FUNCTION_BLOCK FIFO_StatsAggregate
VAR_INPUT
	Overwrite: BOOL;
	pFIFO: POINTER TO StatsAggregateFIFOBuffer;
	in: StatsAggregateRecord;
END_VAR

VAR_OUTPUT
	Err: BOOL;
	Count: DINT;
	Full: BOOL;
	out: StatsAggregateRecord;
END_VAR

VAR
	Head	: UDINT;
	Tail	: UDINT;
	Idx		: UDINT;
END_VAR

ACTION INIT:
Idx := pFIFO^.Size * SIZEOF(in);
MEMSET(ADR(pFIFO^.Buffer[0]), 0, Idx);
MEMSET(ADR(in), 0, SIZEOF(in));
MEMSET(ADR(out), 0, SIZEOF(out));
Count := 0;
Head := 0;
Tail := 0;
Full := 0;
Err := 0;
END_ACTION

ACTION LOAD:
Err := 0;
IF (Full AND Overwrite) OR NOT Full THEN
	pFIFO^.Buffer[Head] := in;
	Head := Head + 1;
	IF Head = pFIFO^.Size THEN
		Head := 0;
	END_IF
	IF Full THEN
		Tail := Tail + 1;
		IF Tail = pFIFO^.Size THEN
			Tail := 0;
		END_IF
	ELSE
		Count := Count + 1;
	END_IF
ELSE
	Err := 1;
END_IF
Full := (Head = Tail);
END_ACTION

ACTION PEEK:
Err := 0;
IF Full OR (Tail <> Head) THEN
	out := pFIFO^.Buffer[Head];
ELSE
	Err := 1; (*fifo is empty*)
END_IF
END_ACTION

ACTION PEEKLAST:
Err := 0;
IF Full OR (Tail <> Head) THEN
	out := pFIFO^.Buffer[Tail];
ELSE
	Err := 1; (*fifo is empty*)
END_IF
END_ACTION

ACTION UNLOAD:
Err := 0;
IF NOT Full AND (Head = Tail) THEN
	(*empty*)
	Err := 1;
ELSE
	out := pFIFO^.Buffer[Tail];
	MEMSET(ADR(pFIFO^.Buffer[Tail]), 0, SIZEOF (in));
	Tail := Tail + 1;
	Count := Count - 1;
	IF Tail = pFIFO^.Size THEN
		Tail := 0;
	END_IF
	Full := 0;
END_IF
END_ACTION

END_FUNCTION_BLOCK

(* stored: Version 1.1.0.1, ProductVersion 3.1.4024.9
   POU FIFO_StatsAggregate: Id {b7a99786-5d16-492a-8d8e-dd8c9b51930a}, SpecialFunc None
   Action INIT: Id {65934f49-a995-4b17-879a-02fcbc7714ad}
   Action LOAD: Id {621ab890-1cdd-41a1-a878-1ba9f75117f1}
   Action PEEK: Id {4ff64e57-926d-4c21-b544-0a69b0659063}
   Action PEEKLAST: Id {97c8f260-51d0-48b6-b463-4c007ca88bf0}
   Action UNLOAD: Id {6fdc46b5-329a-45b3-a299-0f6712f0bb1b} *)
